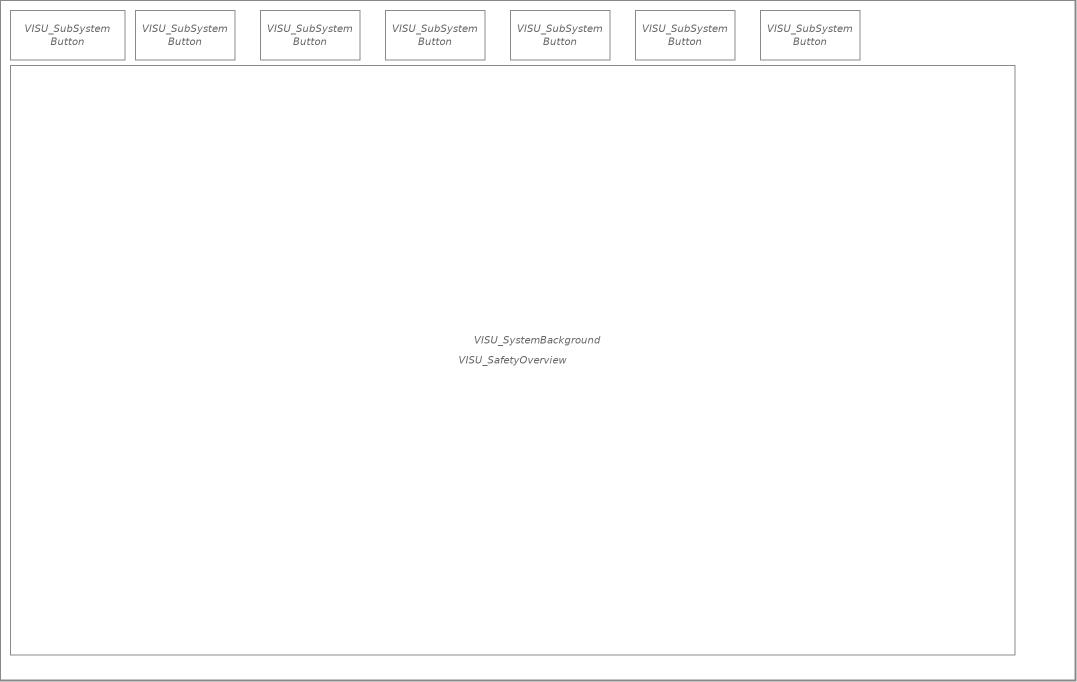
VISUALIZATION VISU_Safety  // 1077x682
VAR_IN_OUT
	ref : Safety;
    widget : SafetyWidget;
END_VAR
    Frame (0,0 1075x680)
        shows VISU_SystemBackground(color := widget.actualStatus.color)
    Frame (10,65 1005x590)
        shows VISU_SafetyOverview(ref := ref, widget := widget)
        shows VISU_SafetyEmergencyStops(ref := ref.parts.emergencyStops, widget := widget.emergencyStops)
        shows VISU_SafetyHydraulics(ref := ref.parts.hydraulics, widget := widget.hydraulics)
        shows VISU_SafetyDomeAccess(ref := ref.parts.domeAccess, widget := widget.domeAccess)
        shows VISU_SafetyMotionBlocking(ref := ref.parts.motionBlocking, ref_hydraulics := ref.parts.hydraulics, ref_emergencyStops := ref.parts.emergencyStops, ref_domeAccess := ref.parts.domeAccess, widget := widget.motionBlocking)
        shows VISU_SafetyIO(ref := ref.parts.io, widget := widget.io)
        shows VISU_SafetyConfig(editable := ref.editableConfig, active := ref.config, mgr := ref.parts.configManager, mgrWidget := widget.configManager, widget := widget)
        p701045219: ref.editableConfig
        p2690442461: ref.config
    Frame (10,10 115x50)
        shows VISU_SubSystemButton(widget := widget.button_overview)
        OnMouseClick: FrameSelectionChange Selection=SelectedFrame=b1e9e4b0-bf3d-440f-90c5-cb513105ccf1, GlobSel=AssignType=Directly, SelType=Locally
        OnMouseClick: execute { widget.activeTab := SafetyTabs.OVERVIEW; }
    Frame (635,10 100x50)
        shows VISU_SubSystemButton(widget := widget.button_io)
        OnMouseClick: FrameSelectionChange Selection=SelectedFrame=b1e9e4b0-bf3d-440f-90c5-cb513105ccf1, Selection=5, GlobSel=AssignType=Directly, SelType=Locally
        OnMouseClick: execute { widget.activeTab := SafetyTabs.IO; }
    Frame (760,10 100x50)
        shows VISU_SubSystemButton(widget := widget.button_config)
        OnMouseClick: FrameSelectionChange Selection=SelectedFrame=b1e9e4b0-bf3d-440f-90c5-cb513105ccf1, Selection=6, GlobSel=AssignType=Directly, SelType=Locally
        OnMouseClick: execute { widget.activeTab := SafetyTabs.CONFIG; }
    Frame (135,10 100x50)
        shows VISU_SubSystemButton(widget := widget.button_emergencyStops)
        OnMouseClick: FrameSelectionChange Selection=SelectedFrame=b1e9e4b0-bf3d-440f-90c5-cb513105ccf1, Selection=1, GlobSel=AssignType=Directly, SelType=Locally
        OnMouseClick: execute { widget.activeTab := SafetyTabs.EMERGENCY_STOPS; }
    Frame (260,10 100x50)
        shows VISU_SubSystemButton(widget := widget.button_hydraulics)
        OnMouseClick: FrameSelectionChange Selection=SelectedFrame=b1e9e4b0-bf3d-440f-90c5-cb513105ccf1, Selection=2, GlobSel=AssignType=Directly, SelType=Locally
        OnMouseClick: execute { widget.activeTab := SafetyTabs.HYDRAULICS; }
    Frame (510,10 100x50)
        shows VISU_SubSystemButton(widget := widget.button_motionBlocking)
        OnMouseClick: FrameSelectionChange Selection=SelectedFrame=b1e9e4b0-bf3d-440f-90c5-cb513105ccf1, Selection=4, GlobSel=AssignType=Directly, SelType=Locally
        OnMouseClick: execute { widget.activeTab := SafetyTabs.MOTION_BLOCKING; }
    Frame (385,10 100x50)
        shows VISU_SubSystemButton(widget := widget.button_domeAccess)
        OnMouseClick: FrameSelectionChange Selection=SelectedFrame=b1e9e4b0-bf3d-440f-90c5-cb513105ccf1, Selection=3, GlobSel=AssignType=Directly, SelType=Locally
        OnMouseClick: execute { widget.activeTab := SafetyTabs.DOME_ACCESS; }
END_VISUALIZATION

(* stored: Version 1.1.0.1, ProductVersion 3.1.4019.2
   Visu VISU_Safety: Id {d9363c50-912c-4208-85b6-a3f6322be761} *)
